PROGRAM MAIN
VAR
	fbArray:Task1;
	fbArrayCheck:Task2;
	fbPage:Task3_GLV_HMI;
END_VAR

fbArray();
fbArrayCheck();
fbPage();

END_PROGRAM

(* stored: Version 1.1.0.1, ProductVersion 3.1.4024.13
   POU MAIN: Id {0b88644e-bdd6-4b1d-9d5c-bb337beb1445}, SpecialFunc None *)
